% RSLogix 500 project OSR.RSS, saved by version 8.30.00.16 %
PROJECT "OSR"    % processor: Bul.1763 MicroLogix 1100 Series B %

PROGRAM FILES
  LAD 2   2 rungs

DATA FILES
  O0 OUTPUT  4 elements
  I1 INPUT  6 elements
  S2 STATUS  66 elements
  B3 BINARY  1 elements
  T4 TIMER  1 elements
  C5 COUNTER  1 elements
  R6 CONTROL  1 elements
  N7 INTEGER  1 elements
  F8 FLOAT  1 elements

LADDER 2
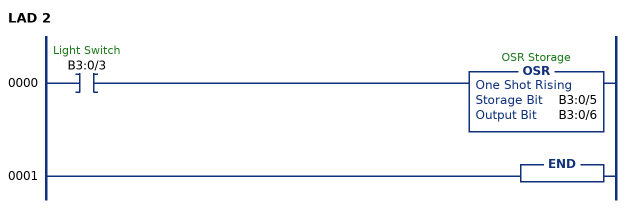
% Rung: 0 %  % edit flag set %
SOR XIC B3:0/3 OSR B3:0/5 B3:0/6 EOR
%   B3:0/3  "Light Switch" %
%   B3:0/5  "OSR Storage" %
% Rung: 1 %
SOR END EOR
